Staubli VAL3: splitUp.pgx

program splitUp(point x_pSphere1, point x_pSphere2, point x_pSphere3, point x_pSphere4)
begin
  //-----------------------------------------------------------------------
  //Header begin
  //Description of program
  //  This program calculates the sphere.
  //
  //Input parameters
  //  point x_pSphere1 to point x_pSphere4 :
  //
  //Traceability
  //  Creation : 07-04-08 - f.Rob
  //  Used without modification for SLAC  KN 17aug2009
  //Header end
  //-----------------------------------------------------------------------

  trSphere[0]=x_pSphere1.trsf
  trSphere[1]=x_pSphere2.trsf
  trSphere[2]=x_pSphere3.trsf
  trSphere[3]=x_pSphere4.trsf
  nS1[1]=trSphere[0].x
  nS1[2]=trSphere[0].y
  nS1[3]=trSphere[0].z
  nS2[1]=trSphere[1].x
  nS2[2]=trSphere[1].y
  nS2[3]=trSphere[1].z
  nS3[1]=trSphere[2].x
  nS3[2]=trSphere[2].y
  nS3[3]=trSphere[2].z
  nS4[1]=trSphere[3].x
  nS4[2]=trSphere[3].y
  nS4[3]=trSphere[3].z
end
